{attribute 'GeneratedUsingTerminal: EK1122-0000-0018'}
{attribute addProperty BoxType "EK1122-0000-0018"}
{attribute addProperty Id "Beckhoff_ER8xxxsub_EK1100EK1100_AB5A94672A_0001_ER8309_1022_0018ER8309_35A864DD70"}
{attribute addProperty CRC "3517236470"}
{attribute addProperty Size "72"}
TYPE Beckhoff_ER8xxxEK1122_D1A4C4F6 EXTENDS EK1122_AB5A9467 :
STRUCT
	{attribute addProperty Name "Beckhoff_ER8xxxsub_EK1100"}
	Beckhoff_ER8xxxsub_EK1100 : EK1100_AB5A9467;
	{attribute addProperty Name "A_0001_ER8309_1022_0018"}
	A_0001_ER8309_1022_0018 : ER8309_35A864DD;
END_STRUCT
END_TYPE

(* stored: Version 1.2.0.0, ProductVersion 3.1.4024.9
   DUT Beckhoff_ER8xxxEK1122_D1A4C4F6: Id {926e378a-bf74-4b05-bd81-5e65364183c8} *)
